(* IEC 61131-3 sources: DNS/HMIRemote (part 2) *)

			(* *** REFRESHING PARENT BACKGROUND ITEMS *** *)

		END_IF;

		(* Unlocking the video *)
		res := Video_Unlock( res );

		(* Suspending the task *)
		res := Video_Sleep( 50 );

	UNTIL pagID <> 16#00
	END_REPEAT;

END_FUNCTION_BLOCK

FUNCTION_BLOCK RefrSETUP_PR2

	VAR_EXTERNAL
	guiCallStack : ARRAY[ 0..9 ] OF UINT;
	giStackPtr : INT;
	fbSETUP_PR2String_19 : Static01;
	fbSETUP_PR2String_20 : Static01;
	fbSETUP_PR2Edit_21 : EditBox01;
	fbSETUP_PR2Edit_22 : EditBox01;
	$waitRefresh : BOOL;
	END_VAR

	VAR
	res : USINT;
	pagID : UINT;
	n : USINT;
	iSP : INT;
	pDC : UDINT;
	rx1 : UINT;
	ry1 : UINT;
	rx2 : UINT;
	ry2 : UINT;
	END_VAR

	{CODE:ST}

	REPEAT

		(* Locking the video *)
		res := Video_Lock( res );

		(* Testing if page has changed *)
		pagID := guiCallStack[ giStackPtr ];

		IF pagID = 16#01 THEN

			(* the refresh task is arrived *)
			$waitRefresh := FALSE;

			(* *** REFRESH PAGE CONTROLS *** *)
			IF fbSETUP_PR2Edit_21.accMode <> kACS_MODIFY THEN
				fbSETUP_PR2Edit_21();
			END_IF;
			IF fbSETUP_PR2Edit_22.accMode <> kACS_MODIFY THEN
				fbSETUP_PR2Edit_22();
			END_IF;

			(* *** REFRESHING BACKGROUND ITEMS *** *)
			(* Cursor across the call stack *)
			iSP := giStackPtr;

			(* *** REFRESHING PARENT BACKGROUND ITEMS *** *)

		END_IF;

		(* Unlocking the video *)
		res := Video_Unlock( res );

		(* Suspending the task *)
		res := Video_Sleep( 50 );

	UNTIL pagID <> 16#01
	END_REPEAT;

END_FUNCTION_BLOCK

FUNCTION_BLOCK RefrSETUP_PR1

	VAR_EXTERNAL
	guiCallStack : ARRAY[ 0..9 ] OF UINT;
	giStackPtr : INT;
	fbSETUP_PR1String_1 : Static01;
	fbSETUP_PR1String_3 : Static01;
	fbSETUP_PR1String_19 : Static01;
	fbSETUP_PR1String_20 : Static01;
	fbSETUP_PR1Edit_17 : EditBox01;
	fbSETUP_PR1Edit_18 : EditBox01;
	fbSETUP_PR1Edit_21 : EditBox01;
	fbSETUP_PR1Edit_22 : EditBox01;
	$waitRefresh : BOOL;
	END_VAR

	VAR
	res : USINT;
	pagID : UINT;
	n : USINT;
	iSP : INT;
	pDC : UDINT;
	rx1 : UINT;
	ry1 : UINT;
	rx2 : UINT;
	ry2 : UINT;
	END_VAR

	{CODE:ST}

	REPEAT

		(* Locking the video *)
		res := Video_Lock( res );

		(* Testing if page has changed *)
		pagID := guiCallStack[ giStackPtr ];

		IF pagID = 16#02 THEN

			(* the refresh task is arrived *)
			$waitRefresh := FALSE;

			(* *** REFRESH PAGE CONTROLS *** *)
			IF fbSETUP_PR1Edit_17.accMode <> kACS_MODIFY THEN
				fbSETUP_PR1Edit_17();
			END_IF;
			IF fbSETUP_PR1Edit_18.accMode <> kACS_MODIFY THEN
				fbSETUP_PR1Edit_18();
			END_IF;
			IF fbSETUP_PR1Edit_21.accMode <> kACS_MODIFY THEN
				fbSETUP_PR1Edit_21();
			END_IF;
			IF fbSETUP_PR1Edit_22.accMode <> kACS_MODIFY THEN
				fbSETUP_PR1Edit_22();
			END_IF;

			(* *** REFRESHING BACKGROUND ITEMS *** *)
			(* Cursor across the call stack *)
			iSP := giStackPtr;

			(* *** REFRESHING PARENT BACKGROUND ITEMS *** *)

		END_IF;

		(* Unlocking the video *)
		res := Video_Unlock( res );

		(* Suspending the task *)
		res := Video_Sleep( 50 );

	UNTIL pagID <> 16#02
	END_REPEAT;

END_FUNCTION_BLOCK

FUNCTION_BLOCK RefrSETUP_RS2

	VAR_EXTERNAL
	guiCallStack : ARRAY[ 0..9 ] OF UINT;
	giStackPtr : INT;
	fbSETUP_RS2String_1 : Static01;
	fbSETUP_RS2String_3 : Static01;
	fbSETUP_RS2String_5 : Static01;
	fbSETUP_RS2String_7 : Static01;
	fbSETUP_RS2String_9 : Static01;
	fbSETUP_RS2String_11 : Static01;
	fbSETUP_RS2Edit_12 : EditBox01;
	fbSETUP_RS2Edit_13 : EditBox01;
	fbSETUP_RS2Edit_14 : EditBox01;
	fbSETUP_RS2Edit_15 : EditBox01;
	fbSETUP_RS2Edit_16 : EditBox01;
	fbSETUP_RS2Edit_17 : EditBox01;
	$waitRefresh : BOOL;
	END_VAR

	VAR
	res : USINT;
	pagID : UINT;
	n : USINT;
	iSP : INT;
	pDC : UDINT;
	rx1 : UINT;
	ry1 : UINT;
	rx2 : UINT;
	ry2 : UINT;
	END_VAR

	{CODE:ST}

	REPEAT

		(* Locking the video *)
		res := Video_Lock( res );

		(* Testing if page has changed *)
		pagID := guiCallStack[ giStackPtr ];

		IF pagID = 16#03 THEN

			(* the refresh task is arrived *)
			$waitRefresh := FALSE;

			(* *** REFRESH PAGE CONTROLS *** *)
			IF fbSETUP_RS2Edit_12.accMode <> kACS_MODIFY THEN
				fbSETUP_RS2Edit_12();
			END_IF;
			IF fbSETUP_RS2Edit_13.accMode <> kACS_MODIFY THEN
				fbSETUP_RS2Edit_13();
			END_IF;
			IF fbSETUP_RS2Edit_14.accMode <> kACS_MODIFY THEN
				fbSETUP_RS2Edit_14();
			END_IF;
			IF fbSETUP_RS2Edit_15.accMode <> kACS_MODIFY THEN
				fbSETUP_RS2Edit_15();
			END_IF;
			IF fbSETUP_RS2Edit_16.accMode <> kACS_MODIFY THEN
				fbSETUP_RS2Edit_16();
			END_IF;
			IF fbSETUP_RS2Edit_17.accMode <> kACS_MODIFY THEN
				fbSETUP_RS2Edit_17();
			END_IF;

			(* *** REFRESHING BACKGROUND ITEMS *** *)
			(* Cursor across the call stack *)
			iSP := giStackPtr;

			(* *** REFRESHING PARENT BACKGROUND ITEMS *** *)

		END_IF;

		(* Unlocking the video *)
		res := Video_Unlock( res );

		(* Suspending the task *)
		res := Video_Sleep( 50 );

	UNTIL pagID <> 16#03
	END_REPEAT;

END_FUNCTION_BLOCK

FUNCTION_BLOCK RefrPressure_page

	VAR_EXTERNAL
	guiCallStack : ARRAY[ 0..9 ] OF UINT;
	giStackPtr : INT;
	fbPressure_pageString_1 : Static01;
	fbPressure_pageString_3 : Static01;
	fbPressure_pageString_5 : Static01;
	fbPressure_pageString_7 : Static01;
	fbPressure_pageEdit_8 : EditBox01;
	fbPressure_pageEdit_9 : EditBox01;
	fbPressure_pageEdit_10 : EditBox01;
	fbPressure_pageEdit_11 : EditBox01;
	fbPressure_pageEdit_12 : EditBox01;
	$waitRefresh : BOOL;
	END_VAR

	VAR
	res : USINT;
	pagID : UINT;
	n : USINT;
	iSP : INT;
	pDC : UDINT;
	rx1 : UINT;
	ry1 : UINT;
	rx2 : UINT;
	ry2 : UINT;
	END_VAR

	{CODE:ST}

	REPEAT

		(* Locking the video *)
		res := Video_Lock( res );

		(* Testing if page has changed *)
		pagID := guiCallStack[ giStackPtr ];

		IF pagID = 16#04 THEN

			(* the refresh task is arrived *)
			$waitRefresh := FALSE;

			(* *** REFRESH PAGE CONTROLS *** *)
			fbPressure_pageEdit_8();
			fbPressure_pageEdit_9();
			fbPressure_pageEdit_10();
			fbPressure_pageEdit_11();
			fbPressure_pageEdit_12();

			(* *** REFRESHING BACKGROUND ITEMS *** *)
			(* Cursor across the call stack *)
			iSP := giStackPtr;

			(* *** REFRESHING PARENT BACKGROUND ITEMS *** *)

		END_IF;

		(* Unlocking the video *)
		res := Video_Unlock( res );

		(* Suspending the task *)
		res := Video_Sleep( 50 );

	UNTIL pagID <> 16#04
	END_REPEAT;

END_FUNCTION_BLOCK

FUNCTION_BLOCK RefrMenu

	VAR_EXTERNAL
	guiCallStack : ARRAY[ 0..9 ] OF UINT;
	giStackPtr : INT;
	fbMenuButton_1 : Button02;
	fbMenuButton_2 : Button02;
	$waitRefresh : BOOL;
	END_VAR

	VAR
	res : USINT;
	pagID : UINT;
	n : USINT;
	iSP : INT;
	pDC : UDINT;
	rx1 : UINT;
	ry1 : UINT;
	rx2 : UINT;
	ry2 : UINT;
	END_VAR

	{CODE:ST}

	REPEAT

		(* Locking the video *)
		res := Video_Lock( res );

		(* Testing if page has changed *)
		pagID := guiCallStack[ giStackPtr ];

		IF pagID = 16#05 THEN

			(* the refresh task is arrived *)
			$waitRefresh := FALSE;

			(* *** REFRESH PAGE CONTROLS *** *)

			(* *** REFRESHING BACKGROUND ITEMS *** *)
			(* Cursor across the call stack *)
			iSP := giStackPtr;

			(* *** REFRESHING PARENT BACKGROUND ITEMS *** *)

		END_IF;

		(* Unlocking the video *)
		res := Video_Unlock( res );

		(* Suspending the task *)
		res := Video_Sleep( 50 );

	UNTIL pagID <> 16#05
	END_REPEAT;

END_FUNCTION_BLOCK

FUNCTION_BLOCK RefrSETUP_IP

	VAR_EXTERNAL
	guiCallStack : ARRAY[ 0..9 ] OF UINT;
	giStackPtr : INT;
	fbSETUP_IPString_1 : Static01;
	fbSETUP_IPString_6 : Static01;
	fbSETUP_IPString_11 : Static01;
	fbSETUP_IPString_16 : Static01;
	fbSETUP_IPEdit_2 : EditBox01;
	fbSETUP_IPEdit_3 : EditBox01;
	fbSETUP_IPEdit_4 : EditBox01;
	fbSETUP_IPEdit_5 : EditBox01;
	fbSETUP_IPEdit_7 : EditBox01;
	fbSETUP_IPEdit_8 : EditBox01;
	fbSETUP_IPEdit_9 : EditBox01;
	fbSETUP_IPEdit_10 : EditBox01;
	fbSETUP_IPEdit_12 : EditBox01;
	fbSETUP_IPEdit_13 : EditBox01;
	fbSETUP_IPEdit_14 : EditBox01;
	fbSETUP_IPEdit_15 : EditBox01;
	fbSETUP_IPEdit_17 : EditBox01;
	fbSETUP_IPEdit_18 : EditBox01;
	fbSETUP_IPEdit_19 : EditBox01;
	fbSETUP_IPEdit_20 : EditBox01;
	$waitRefresh : BOOL;
	END_VAR

	VAR
	res : USINT;
	pagID : UINT;
	n : USINT;
	iSP : INT;
	pDC : UDINT;
	rx1 : UINT;
	ry1 : UINT;
	rx2 : UINT;
	ry2 : UINT;
	END_VAR

	{CODE:ST}

	REPEAT

		(* Locking the video *)
		res := Video_Lock( res );

		(* Testing if page has changed *)
		pagID := guiCallStack[ giStackPtr ];

		IF pagID = 16#06 THEN

			(* the refresh task is arrived *)
			$waitRefresh := FALSE;

			(* *** REFRESH PAGE CONTROLS *** *)
			IF fbSETUP_IPEdit_2.accMode <> kACS_MODIFY THEN
				fbSETUP_IPEdit_2();
			END_IF;
			IF fbSETUP_IPEdit_3.accMode <> kACS_MODIFY THEN
				fbSETUP_IPEdit_3();
			END_IF;
			IF fbSETUP_IPEdit_4.accMode <> kACS_MODIFY THEN
				fbSETUP_IPEdit_4();
			END_IF;
			IF fbSETUP_IPEdit_5.accMode <> kACS_MODIFY THEN
				fbSETUP_IPEdit_5();
			END_IF;
			IF fbSETUP_IPEdit_7.accMode <> kACS_MODIFY THEN
				fbSETUP_IPEdit_7();
			END_IF;
			IF fbSETUP_IPEdit_8.accMode <> kACS_MODIFY THEN
				fbSETUP_IPEdit_8();
			END_IF;
			IF fbSETUP_IPEdit_9.accMode <> kACS_MODIFY THEN
				fbSETUP_IPEdit_9();
			END_IF;
			IF fbSETUP_IPEdit_10.accMode <> kACS_MODIFY THEN
				fbSETUP_IPEdit_10();
			END_IF;
			IF fbSETUP_IPEdit_12.accMode <> kACS_MODIFY THEN
				fbSETUP_IPEdit_12();
			END_IF;
			IF fbSETUP_IPEdit_13.accMode <> kACS_MODIFY THEN
				fbSETUP_IPEdit_13();
			END_IF;
			IF fbSETUP_IPEdit_14.accMode <> kACS_MODIFY THEN
				fbSETUP_IPEdit_14();
			END_IF;
			IF fbSETUP_IPEdit_15.accMode <> kACS_MODIFY THEN
				fbSETUP_IPEdit_15();
			END_IF;
			IF fbSETUP_IPEdit_17.accMode <> kACS_MODIFY THEN
				fbSETUP_IPEdit_17();
			END_IF;
			IF fbSETUP_IPEdit_18.accMode <> kACS_MODIFY THEN
				fbSETUP_IPEdit_18();
			END_IF;
			IF fbSETUP_IPEdit_19.accMode <> kACS_MODIFY THEN
				fbSETUP_IPEdit_19();
			END_IF;
			IF fbSETUP_IPEdit_20.accMode <> kACS_MODIFY THEN
				fbSETUP_IPEdit_20();
			END_IF;

			(* *** REFRESHING BACKGROUND ITEMS *** *)
			(* Cursor across the call stack *)
			iSP := giStackPtr;

			(* *** REFRESHING PARENT BACKGROUND ITEMS *** *)

		END_IF;

		(* Unlocking the video *)
		res := Video_Unlock( res );

		(* Suspending the task *)
		res := Video_Sleep( 50 );

	UNTIL pagID <> 16#06
	END_REPEAT;

END_FUNCTION_BLOCK

FUNCTION_BLOCK RefrSETUP

	VAR_EXTERNAL
	guiCallStack : ARRAY[ 0..9 ] OF UINT;
	giStackPtr : INT;
	fbSETUPButton_1 : Button02;
	fbSETUPButton_2 : Button02;
	fbSETUPButton_3 : Button02;
	fbSETUPButton_4 : Button02;
	fbSETUPButton_5 : Button02;
	fbSETUPButton_6 : Button02;
	$waitRefresh : BOOL;
	END_VAR

	VAR
	res : USINT;
	pagID : UINT;
	n : USINT;
	iSP : INT;
	pDC : UDINT;
	rx1 : UINT;
	ry1 : UINT;
	rx2 : UINT;
	ry2 : UINT;
	END_VAR

	{CODE:ST}

	REPEAT

		(* Locking the video *)
		res := Video_Lock( res );

		(* Testing if page has changed *)
		pagID := guiCallStack[ giStackPtr ];

		IF pagID = 16#07 THEN

			(* the refresh task is arrived *)
			$waitRefresh := FALSE;

			(* *** REFRESH PAGE CONTROLS *** *)

			(* *** REFRESHING BACKGROUND ITEMS *** *)
			(* Cursor across the call stack *)
			iSP := giStackPtr;

			(* *** REFRESHING PARENT BACKGROUND ITEMS *** *)

		END_IF;

		(* Unlocking the video *)
		res := Video_Unlock( res );

		(* Suspending the task *)
		res := Video_Sleep( 50 );

	UNTIL pagID <> 16#07
	END_REPEAT;

END_FUNCTION_BLOCK

FUNCTION_BLOCK RefrSETUP_RS1

	VAR_EXTERNAL
	guiCallStack : ARRAY[ 0..9 ] OF UINT;
	giStackPtr : INT;
	fbSETUP_RS1String_1 : Static01;
	fbSETUP_RS1String_3 : Static01;
	fbSETUP_RS1String_5 : Static01;
	fbSETUP_RS1String_7 : Static01;
	fbSETUP_RS1String_9 : Static01;
	fbSETUP_RS1String_11 : Static01;
	fbSETUP_RS1Edit_2 : EditBox01;
	fbSETUP_RS1Edit_4 : EditBox01;
	fbSETUP_RS1Edit_6 : EditBox01;
	fbSETUP_RS1Edit_8 : EditBox01;
	fbSETUP_RS1Edit_10 : EditBox01;
	fbSETUP_RS1Edit_12 : EditBox01;
	$waitRefresh : BOOL;
	END_VAR

	VAR
	res : USINT;
	pagID : UINT;
	n : USINT;
	iSP : INT;
	pDC : UDINT;
	rx1 : UINT;
	ry1 : UINT;
	rx2 : UINT;
	ry2 : UINT;
	END_VAR

	{CODE:ST}

	REPEAT

		(* Locking the video *)
		res := Video_Lock( res );

		(* Testing if page has changed *)
		pagID := guiCallStack[ giStackPtr ];

		IF pagID = 16#08 THEN

			(* the refresh task is arrived *)
			$waitRefresh := FALSE;

			(* *** REFRESH PAGE CONTROLS *** *)
			IF fbSETUP_RS1Edit_2.accMode <> kACS_MODIFY THEN
				fbSETUP_RS1Edit_2();
			END_IF;
			IF fbSETUP_RS1Edit_4.accMode <> kACS_MODIFY THEN
				fbSETUP_RS1Edit_4();
			END_IF;
			IF fbSETUP_RS1Edit_6.accMode <> kACS_MODIFY THEN
				fbSETUP_RS1Edit_6();
			END_IF;
			IF fbSETUP_RS1Edit_8.accMode <> kACS_MODIFY THEN
				fbSETUP_RS1Edit_8();
			END_IF;
			IF fbSETUP_RS1Edit_10.accMode <> kACS_MODIFY THEN
				fbSETUP_RS1Edit_10();
			END_IF;
			IF fbSETUP_RS1Edit_12.accMode <> kACS_MODIFY THEN
				fbSETUP_RS1Edit_12();
			END_IF;

			(* *** REFRESHING BACKGROUND ITEMS *** *)
			(* Cursor across the call stack *)
			iSP := giStackPtr;

			(* *** REFRESHING PARENT BACKGROUND ITEMS *** *)

		END_IF;

		(* Unlocking the video *)
		res := Video_Unlock( res );

		(* Suspending the task *)
		res := Video_Sleep( 50 );

	UNTIL pagID <> 16#08
	END_REPEAT;

END_FUNCTION_BLOCK

	(***************************)
	(*                         *)
	(* PARAMETER  FUN. BLOCKS  *)
	(*                         *)
	(***************************)

	(***************************)
	(*                         *)
	(*   PROC FUNCTIONS        *)
	(*                         *)
	(***************************)
